PROGRAM PRG_MethodReportWriter
VAR
	fbJsonWriter    : FB_JsonSaxWriter;
    eState          : (STATE_IDLE, STATE_START_REPORT_OBJECT, STATE_ADD_REPORT_INFO, STATE_ADD_CALIBRATION_INFO, STATE_START_DATA_ARRAY, STATE_ADD_DATA_LOOP, STATE_END_DATA_ARRAY, STATE_END_REPORT_OBJECT, STATE_COPY_DOCUMENT, STATE_DONE);
	nDataIndex      : INT := 1;
END_VAR

gvl_report.stReportHead.fileName:= PRG_CreateJsonFile.sFileName;

CASE eState OF
    STATE_IDLE:
        IF gvl_report.bBuildMR THEN
            gvl_report.bBuildMR := FALSE;
            fbJsonWriter.ResetDocument();
            nDataIndex := 1;
            eState := STATE_START_REPORT_OBJECT;
        END_IF

    STATE_START_REPORT_OBJECT:
        fbJsonWriter.StartObject(); (* { *)
        eState := STATE_ADD_REPORT_INFO;
    
    STATE_ADD_REPORT_INFO:
        fbJsonWriter.AddKey('reportInfo');
        fbJsonWriter.StartObject(); (* { *)
            fbJsonWriter.AddKeyString('reportName', gvl_report.stReportHead.reportName);
            fbJsonWriter.AddKeyString('reoportSubName', 'Method Report');
            fbJsonWriter.AddKeyString('reportDate', gvl_report.stReportHead.reportDate);
            fbJsonWriter.AddKeyString('systemID', gvl_report.stReportHead.systemID);
            fbJsonWriter.AddKeyString('databaseName', gvl_report.stReportHead.databaseName);
            fbJsonWriter.AddKeyString('page', gvl_report.stReportHead.page);
            fbJsonWriter.AddKeyString('printedBy', gvl_report.stReportHead.printedBy);
			fbJsonWriter.AddKeyString('fileName', gvl_report.stReportHead.fileName);
        fbJsonWriter.EndObject(); (* } *)
        eState := STATE_ADD_CALIBRATION_INFO;

    STATE_ADD_CALIBRATION_INFO:
        fbJsonWriter.AddKey('parametersInfo');
        fbJsonWriter.StartObject(); (* { *)
            fbJsonWriter.AddKeyString('methodName', GVL_Report.stParameter_MR.methodName);
			fbJsonWriter.AddKeyNumber('revision', DINT_TO_UDINT(GVL_Report.stParameter_MR.revision));
            fbJsonWriter.AddKeyString('createdBy', GVL_Report.stParameter_MR.createdBy);
			fbJsonWriter.AddKeyString('createdDate', GVL_Report.stParameter_MR.createdDate);
				fbJsonWriter.AddKey('stepParameters');
				fbJsonWriter.StartObject();
				fbJsonWriter.AddKeyNumber('solv_R1', DINT_TO_UDINT(GVL_Report.stParameter_MR.solv_R1));
				fbJsonWriter.AddKeyNumber('solv_R2', DINT_TO_UDINT(GVL_Report.stParameter_MR.solv_R2));
				fbJsonWriter.AddKeyNumber('solv_W1', DINT_TO_UDINT(GVL_Report.stParameter_MR.solv_W1));
				fbJsonWriter.AddKeyNumber('solv_W2', DINT_TO_UDINT(GVL_Report.stParameter_MR.solv_W2));
				fbJsonWriter.AddKeyNumber('stepTime_R1', DINT_TO_UDINT(GVL_Report.stParameter_MR.stepTime_R1));
				fbJsonWriter.AddKeyNumber('stepTime_R2', DINT_TO_UDINT(GVL_Report.stParameter_MR.stepTime_R2));
				fbJsonWriter.AddKeyNumber('stepTime_W1', DINT_TO_UDINT(GVL_Report.stParameter_MR.stepTime_W1));
				fbJsonWriter.AddKeyNumber('stepTime_W2', DINT_TO_UDINT(GVL_Report.stParameter_MR.stepTime_W2));
				fbJsonWriter.AddKeyNumber('stepRpm_R1', DINT_TO_UDINT(GVL_Report.stParameter_MR.stepRpm_R1));
				fbJsonWriter.AddKeyNumber('stepRpm_R2', DINT_TO_UDINT(GVL_Report.stParameter_MR.stepRpm_R2));
				fbJsonWriter.AddKeyNumber('stepRpm_W1', DINT_TO_UDINT(GVL_Report.stParameter_MR.stepRpm_W1));
				fbJsonWriter.AddKeyNumber('stepRpm_W2', DINT_TO_UDINT(GVL_Report.stParameter_MR.stepRpm_W2));
				fbJsonWriter.EndObject();
			fbJsonWriter.AddKeyNumber('soakTime', DINT_TO_UDINT(GVL_Report.stParameter_MR.soakTime));
			fbJsonWriter.AddKeyNumber('agitateTime1', DINT_TO_UDINT(GVL_Report.stParameter_MR.agitateTime1));
			fbJsonWriter.AddKeyNumber('agitateTime2', DINT_TO_UDINT(GVL_Report.stParameter_MR.agitateTime2));
			fbJsonWriter.AddKeyNumber('vialToFill', DINT_TO_UDINT(GVL_Report.stParameter_MR.vialToFill));
            fbJsonWriter.AddKeyLreal('vialPrimeVol', GVL_Report.stParameter_MR.vialPrimeVol);
			fbJsonWriter.AddKeyLreal('vialFillVol1', GVL_Report.stParameter_MR.vialFillVol1);
			fbJsonWriter.AddKeyLreal('vialsFillVol24', GVL_Report.stParameter_MR.vialsFillVol24);
			fbJsonWriter.AddKeyNumber('airDryTime', DINT_TO_UDINT(GVL_Report.stParameter_MR.airDryTime));
            fbJsonWriter.EndObject(); (* } *)
        eState := STATE_START_DATA_ARRAY;

    STATE_START_DATA_ARRAY:
        fbJsonWriter.AddKey('volumeData');
        fbJsonWriter.StartArray(); (* [ *)
        eState := STATE_ADD_DATA_LOOP;

    STATE_ADD_DATA_LOOP:
        (* Loop para adicionar cada objeto do array *)
		FOR nDataIndex := 1 TO SIZEOF(gvl_report.astData_MR) / SIZEOF(gvl_report.astData_MR[1]) - 1 DO
    		IF gvl_report.astData_MR[nDataIndex].stage = '' THEN
        	// If the dateTime string is empty, break the loop
        	// The condition would "stop" here as you want
			eState := STATE_END_DATA_ARRAY;
       	 	EXIT;
   			ELSE
        	// Continue processing data
				IF nDataIndex < SIZEOF(gvl_report.astData_MR) / SIZEOF(gvl_report.astData_MR[1]) THEN
            		fbJsonWriter.StartObject(); (* { *)
                	fbJsonWriter.AddKeyNumber('pump', DINT_TO_UDINT(gvl_report.astData_MR[nDataIndex].pump));
					fbJsonWriter.AddKeyString('stage', gvl_report.astData_MR[nDataIndex].stage);
                	fbJsonWriter.AddKeylReal('rinse1', gvl_report.astData_MR[nDataIndex].rinse1);
                	fbJsonWriter.AddKeylReal('rinse2', gvl_report.astData_MR[nDataIndex].rinse2);
                	fbJsonWriter.AddKeylReal('wash1', gvl_report.astData_MR[nDataIndex].wash1);
                	fbJsonWriter.AddKeylReal('wash2', gvl_report.astData_MR[nDataIndex].wash2);
            		fbJsonWriter.EndObject(); (* } *)
            		//nDataIndex := nDataIndex + 1;
        		ELSE
            		eState := STATE_END_DATA_ARRAY;
        		END_IF
    		END_IF
		END_FOR
        

    STATE_END_DATA_ARRAY:
        fbJsonWriter.EndArray(); (* ] *)
        eState := STATE_END_REPORT_OBJECT;

    STATE_END_REPORT_OBJECT:
        fbJsonWriter.EndObject(); (* } *)
        eState := STATE_COPY_DOCUMENT;

    STATE_COPY_DOCUMENT:
        fbJsonWriter.CopyDocument(GVL_Report.sJsonOutput, SIZEOF(GVL_Report.sJsonOutput));
        eState := STATE_DONE;

    STATE_DONE:
        eState:= STATE_IDLE; (* O JSON está pronto na variável sJsonOutput *)
		GVL_Report.bStartWrite := TRUE;
		;
    
END_CASE

END_PROGRAM

(* stored: Version 1.1.0.1, ProductVersion 3.1.4024.12
   POU PRG_MethodReportWriter: Id {49e75958-969a-4bac-b5e2-9552e123dc81}, SpecialFunc None *)
